Universal Robots PolyScope program: edges.urp

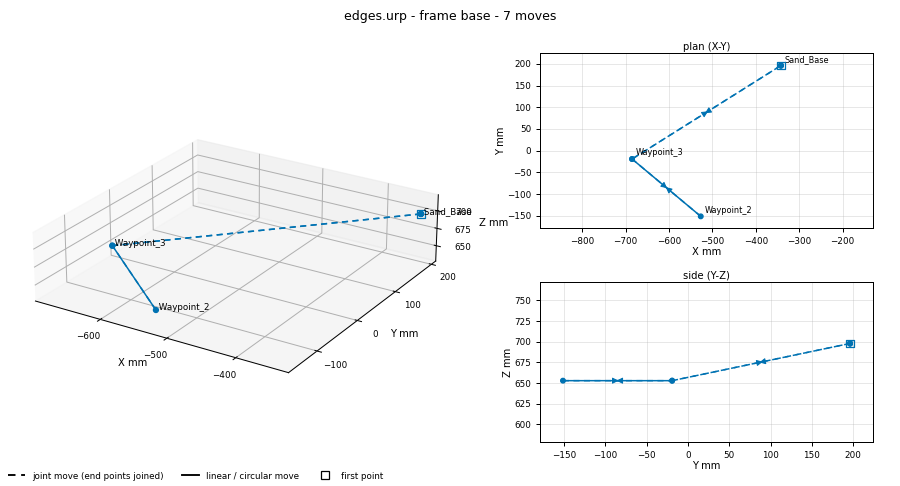
[picture p0: tool path of edges.urp in frame base, 7 of 7 moves have a stored position in this frame; points joined in program order, loops and branches not executed]
Program edges (installation=cube_dev1 directory=/programs/cube createdIn=5.11.5.1010327 lastSavedIn=5.11.5.1010327 robotSerialNumber=20215500677)
Calibrated DH parameters: a=[0.000204, -0.239222, -0.391845, -0.000001, 0.000022, 0]; d=[0.162722, -355.808559, 353.37206, 2.570385, 0.099741, 0.099629]; alpha=[1.571124, 0.000988, 0.008295, 1.568963, -1.570303, 0]; deltaTheta=[0, -0.973091, 7.204745, 0.05153, 0, 0]
Robot Program (runOnlyOnce=true)
  MoveJ speed 120 deg/s, acceleration 120 deg/s^2 (useActiveTCP=false) tcp=SandTCP; feature=Point_1
    Waypoint Sand_Base: TCP in base x=-341.949 y=196.192 z=697.874 mm, rx=0 ry=0 rz=-1.5708 rad; joints [-57.163, -82.73, 107.731, 93.373, -53.983, -132.185] deg; TCP offset x=1.003 y=125.541 z=104.154 mm, rx=-0.7854 ry=0 rz=0 rad; feature pose in base x=-341.965 y=196.202 z=697.85 mm, rx=0 ry=0 rz=-1.5843 rad
  Folder Sand
    MoveL speed 50 mm/s, acceleration 1200 mm/s^2 (useActiveTCP=false) tcp=SandTCP; feature=Base
      MoveDirectionNode (selectedDirection=ZPlus)
        Until TOOL_CONTACT_DETECTION (allowActions=false retraction=0.001 decelerationAcceleration=3 decelerationAngularAcceleration=34.906585)
      URCap Finishing Tool Control (Robotiq_Copilot, Robotiq Inc.) dataModel(ToolOutputNameKey=SanderOn, HackTriggeringContributionIsDefinedMethodKey=true)
    MoveL speed 50 mm/s, acceleration 1200 mm/s^2 (useActiveTCP=true) feature=Base
      Force Simple feature=Base; selection=[0, 0, 1, 0, 0, 0]; wrench=[0, 0, 5, 0, 0, 0]; limitsForce=[0.15, 0.15, 0.15, 1.047198, 1.047198, 1.047198]; limitsMotion=[0.1, 0.1, 0.1, 0.349066, 0.349066, 0.349066]
        MoveDirectionNode (selectedDirection=XMinus)
          Until DISTANCE (allowActions=false deceleration=3 distanceNodeType=BLEND) Distance=0.355; motionParameters(blendRadius=0.025)
        MoveDirectionNode (selectedDirection=YMinus)
          Until DISTANCE (allowActions=false deceleration=3 distanceNodeType=BLEND) Distance=0.355; motionParameters(blendRadius=0.025)
        MoveDirectionNode (selectedDirection=XPlus)
          Until DISTANCE (allowActions=false deceleration=3 distanceNodeType=BLEND) Distance=0.355; motionParameters(blendRadius=0.025)
        MoveDirectionNode (selectedDirection=YPlus)
          Until DISTANCE (allowActions=false deceleration=3 distanceNodeType=STOP) Distance=0.355; motionParameters(blendRadius=0.01)
        URCap Finishing Tool Control (Robotiq_Copilot, Robotiq Inc.) dataModel(FinishingToolStateKey=false, ToolOutputNameKey=SanderOn, HackTriggeringContributionIsDefinedMethodKey=true)
    MoveL speed 90 mm/s, acceleration 1200 mm/s^2 (useActiveTCP=false) tcp=SandTCP; feature=Base
      MoveDirectionNode (selectedDirection=ZMinus)
        Until DISTANCE (allowActions=false deceleration=3 distanceNodeType=BLEND) Distance=0.05; motionParameters(blendRadius=0.003)
  Folder Spray Vert
    MoveJ speed 120 deg/s, acceleration 150 deg/s^2 (useActiveTCP=false) tcp=SprayTCP; feature=Point_1
      Waypoint Spray_Base: TCP in base x=-341.952 y=196.173 z=697.866 mm, rx=0 ry=0 rz=0.0032 rad; joints [-64.094, -80.171, 99.151, 94.355, -50.864, 55.964] deg; TCP offset x=-61.38 y=-97.07 z=93.78 mm, rx=0.6139 ry=0.6139 rz=-1.4822 rad
    MoveL speed 90 mm/s, acceleration 1200 mm/s^2 (useActiveTCP=false) tcp=SprayTCP; feature=Base
      MoveDirectionNode (selectedDirection=ZMinus)
        Until DISTANCE (allowActions=false deceleration=3 distanceNodeType=BLEND) Distance=0.05; motionParameters(blendRadius=0.003)
      Set DigitalOutput pin=digital_out[5]; digitalValue=1
      MoveDirectionNode (selectedDirection=XMinus)
        Until DISTANCE (allowActions=false deceleration=3 distanceNodeType=BLEND) Distance=0.355; motionParameters(blendRadius=0.003)
      MoveDirectionNode (selectedDirection=YMinus)
        Until DISTANCE (allowActions=false deceleration=3 distanceNodeType=BLEND) Distance=0.355; motionParameters(blendRadius=0.003)
      MoveDirectionNode (selectedDirection=XPlus)
        Until DISTANCE (allowActions=false deceleration=3 distanceNodeType=BLEND) Distance=0.355; motionParameters(blendRadius=0.003)
      MoveDirectionNode (selectedDirection=YPlus)
        Until DISTANCE (allowActions=false deceleration=3 distanceNodeType=BLEND) Distance=0.355; motionParameters(blendRadius=0.003)
      Set DigitalOutput pin=digital_out[5]; digitalValue=0
  Folder Spray Horiz
    MoveJ speed 120 deg/s, acceleration 150 deg/s^2 (useActiveTCP=false) tcp=SprayTCP; feature=Point_1
      Waypoint Spray_Base: TCP in base x=-341.952 y=196.173 z=697.866 mm, rx=0 ry=0 rz=0.0032 rad; joints [-64.094, -80.171, 99.151, 94.355, -50.864, 55.964] deg
      Waypoint Waypoint_3: TCP in base x=-684.904 y=-19.185 z=652.836 mm, rx=0.8223 ry=0.8113 rz=-1.4242 rad; joints [-23.453, -71.182, 83.411, -108.112, 76.632, 113.221] deg; TCP offset x=-61.38 y=-97.07 z=93.78 mm, rx=0.6139 ry=0.6139 rz=-1.4822 rad
      Set DigitalOutput pin=digital_out[5]; digitalValue=1
      MoveL speed 100 mm/s, acceleration 1200 mm/s^2 (useActiveTCP=false) tcp=SprayTCP; feature=Point_1
        MoveDirectionNode (selectedDirection=XPlus) feature=Base
          Until DISTANCE (allowActions=false deceleration=3 distanceNodeType=STOP) Distance=0.34; motionParameters(blendRadius=0)
        Set DigitalOutput pin=digital_out[5]; digitalValue=0
        Waypoint Waypoint_2: motionParameters(jointSpeed=1.047198 jointAcceleration=1.396263 cartesianSpeed=0.25 cartesianAcceleration=1.2); TCP in base x=-526.678 y=-151.321 z=652.844 mm, rx=0.0071 ry=1.0472 rz=-0.0122 rad; joints [-3.948, -64.662, 76.505, -116.857, 91.255, 182.817] deg; TCP offset x=-61.38 y=-97.07 z=93.78 mm, rx=0.6139 ry=0.6139 rz=-1.4822 rad
        Set DigitalOutput pin=digital_out[5]; digitalValue=1
        MoveDirectionNode (selectedDirection=YPlus) feature=Base
          Until DISTANCE (allowActions=false deceleration=3 distanceNodeType=STOP) Distance=0.34; motionParameters(blendRadius=0)
        Set DigitalOutput pin=digital_out[5]; digitalValue=0
      MoveJ speed 120 deg/s, acceleration 150 deg/s^2 (useActiveTCP=false) tcp=SprayTCP; feature=Point_1
        Waypoint Waypoint_1: TCP in base x=-684.904 y=-19.185 z=652.833 mm, rx=-0.8086 ry=0.8199 rz=1.4004 rad; joints [2.191, -51.965, 52.949, -91.828, 105.466, -93.13] deg; TCP offset x=-61.38 y=-97.07 z=93.78 mm, rx=0.6139 ry=0.6139 rz=-1.4822 rad
        Set DigitalOutput pin=digital_out[5]; digitalValue=1
      MoveL speed 100 mm/s, acceleration 1200 mm/s^2 (useActiveTCP=true) feature=Base
        MoveDirectionNode (selectedDirection=XPlus) feature=Base
          Until DISTANCE (allowActions=false deceleration=3 distanceNodeType=STOP) Distance=0.34; motionParameters(blendRadius=0)
        Set DigitalOutput pin=digital_out[5]; digitalValue=0
  MoveJ speed 120 deg/s, acceleration 120 deg/s^2 (useActiveTCP=false) tcp=SandTCP; feature=Point_1
    Waypoint Sand_Base: TCP in base x=-341.949 y=196.192 z=697.874 mm, rx=0 ry=0 rz=-1.5708 rad; joints [-57.163, -82.73, 107.731, 93.373, -53.983, -132.185] deg; TCP offset x=1.003 y=125.541 z=104.154 mm, rx=-0.7854 ry=0 rz=0 rad
